Fanuc KAREL source: kt00026.KL

-- PROVISIONAL review KL for V940-1; original PC SHA256 b43a64750f451fabb008d2f221fd70a7a6ac8e4d631161d128a2c5f73c27783c
-- Incomplete behavior may be omitted. Consult companion uncertainty JSON. Do not deploy.
PROGRAM KT00026
%NOLOCKGROUP
VAR
  I2 : INTEGER
  OUT : REAL
-- UNRESOLVED_DECL H1 type=002017
BEGIN
  -- V9_ZERO_TABLE_METADATA_HINT layout=0001; no indexed target words; source/name/runtime held
  -- UNRESOLVED_PC offsets 5-19; opcodes 2E,22,9D,33,B4
  -- UNRESOLVED_PC offsets 24-35; opcodes 2E,23
  -- UNRESOLVED_PC offsets 40-63; opcodes 22,9D,33,B3,21,52,64,23
  -- UNRESOLVED_PC offsets 68-72; opcodes 7F
END KT00026
